KUKA KRL program: PickEsteira.src, PickEsteira.dat

--- PickEsteira.src ---
&ACCESS RVO1
&REL 95
&PARAM DISKPATH = KRC:\R1\Program\MainRoutune\Pick
DEF PickEsteira ( )
   PuxaReceita()
   $Advance=3
   ConfGarra_nowait()

   ;FOLD verifica qual opcao de base para a esteira
      SWITCH PalletAtivo
         CASE 1
            BaseRelativa.X = BaseEsteira1.X + OffsetEsteira1.X
            BaseRelativa.Y = BaseEsteira1.Y + OffsetEsteira1.Y
            BaseRelativa.Z = BaseEsteira1.Z + OffsetEsteira1.Z
            BaseRelativa.A = BaseEsteira1.A + OffsetEsteira1.A
            BaseRelativa.B = BaseEsteira1.B + OffsetEsteira1.B
            BaseRelativa.C = BaseEsteira1.C + OffsetEsteira1.C
         CASE 2
            BaseRelativa.X = BaseEsteira2.X + OffsetEsteira2.X
            BaseRelativa.Y = BaseEsteira2.Y + OffsetEsteira2.Y
            BaseRelativa.Z = BaseEsteira2.Z + OffsetEsteira2.Z
            BaseRelativa.A = BaseEsteira2.A + OffsetEsteira2.A
            BaseRelativa.B = BaseEsteira2.B + OffsetEsteira2.B
            BaseRelativa.C = BaseEsteira2.C + OffsetEsteira2.C
         DEFAULT
            BaseRelativa = NULLFRAME
      ENDSWITCH
   ;ENDFOLD

   ;FOLD PickEsteira de cada receita
      Tpick_esteira()
      XPICK = pick_esteira[PalletAtivo,PickOp]
   ;ENDFOLD

   ;SET BaseRelativa
   $TOOL = TOOL_DATA[1]
   $BASE=BaseRelativa

   ;SET Ponto de pick
   XAPP1PICK = XPICK
   XAPP2PICK = XPICK
   XSAIPICK  = XPICK

   ;Captura o Y da esteira para o ponto de aproximacao
   ;IF (PalletAtivo==1) THEN
   ;   XAPP1PICK.Y = XAPP1PICK.Y - 50
   ;   XAPP2PICK.Y = XAPP2PICK.Y - 50
   ;ENDIF

   ;IF (PalletAtivo==2) THEN
   ;   XAPP1PICK.Y = XAPP1PICK.Y + 50
   ;   XAPP2PICK.Y = XAPP2PICK.Y + 50
   ;ENDIF

   ;FOLD raciocinio do calculo de igualar bases
      ;    ZPick  _      _ ZPlace
      ;           |      |
      ;           |      |
      ;           |      |
      ;           |      - BPlace
      ;           |      |
      ;    BPick  -      |
      ;           |      |
      ;           |      |
      ;             ZERO

      ;ZPick  + BPick  = ZPlace + BPlace

      ;ZPick  = ZPlace + BPlace - BPick
      ;ZPlace = ZPick  + BPick  - BPlace

      ;ALTURATOPO=1800
      ;ZPick  = ALTURATOPO - BPick
      ;ZPlace = ALTURATOPO - BPlace
   ;ENDFOLD

   ;FOLD TOPO DINAMICO IGUALANDO A BASE PLACE COM A DO PICK
      ;Puxa qual o ponto que sera feito o Place
      SetPlacePos()
      ;iguala as bases para obter o Z relativo
      ;ZPick      = ZPlace       +  BPlace                                          - BPick
      XAPP1PICK.Z = XApp1Place.Z + (BasePoint.Z + OffSetPallet.Z + OffsetProduto.Z) - BaseRelativa.Z

      ;Configura a altura de saida do pick
      XSAIPICK.Z = XAPP1PICK.Z

      ;Se o pallet estiver completo o pick eh forcado com a altura MAX
      IF (PalletCompleto==TRUE) THEN
         XAPP1PICK.Z = AlturaPalletCompleto - BaseRelativa.Z
         PalletCompleto=FALSE
      ENDIF

      ;Por seguranca deve garantir que sempre sera acima da altura minima
      ; ZPick2 = ALTURATOPO - BPick
      ; IF (ZPick1 < ZPick2)
      IF (XAPP1PICK.Z<(ALTURATOPO - BaseRelativa.Z)) THEN
         XAPP1PICK.Z = ALTURATOPO - BaseRelativa.Z
      ENDIF
      ;Por seguranca deve garantir que sempre sera acima da altura minima
      IF (XSAIPICK.Z<(ALTURATOPO - BaseRelativa.Z)) THEN
         XSAIPICK.Z  = ALTURATOPO - BaseRelativa.Z
      ENDIF
   ;ENDFOLD

   ;APROXIMA TOPO
   PTP XAPP1PICK C_DIS

   ;CONFIGURA GARRA
   ;ConfGarra()
   ConfGarra_Wait()

   ;APROXIMA DA CAIXA
   LIN XAPP2PICK C_DIS C_DIS

   ;PONTO DE PICK
   LIN XPICK

   ;Fecha Garra
   FechaGarra()

   ;TRAVA/FREIA GARRA
   IF (TravaGarra) THEN
      HomePositionBrake = TRUE
      WorkPositionBrake = FALSE
   ELSE
      HomePositionBrake = FALSE
      WorkPositionBrake = TRUE
   ENDIF

   ;SOBE EM MOVIMENTO RELATIVO
   LIN XSAIPICK

END

--- PickEsteira.dat ---
&ACCESS RVO1
&REL 95
&PARAM DISKPATH = KRC:\R1\Program\MainRoutune\Pick
DEFDAT  PICKESTEIRA
REAL TopoRelativo=707.875305
FRAME RelFrame={X 0.0,Y 0.0,Z 0.0,A 0.0,B 0.0,C 0.0}
FRAME BaseRelativa={X 648.495,Y -1967.36694,Z -56.0000,A 0.0,B 0.0,C 0.0}
DECL E6POS XAPP1PICK={X 491.530762,Y 56.8316116,Z 1968.79492,A 90.0000,B 0.0,C -180.000,S 2,T 34,E1 0.0,E2 0.0,E3 0.0,E4 0.0,E5 0.0,E6 0.0}
DECL E6POS XAPP2PICK={X 491.530762,Y 56.8316116,Z 1343.55737,A 90.0000,B 0.0,C -180.000,S 2,T 34,E1 0.0,E2 0.0,E3 0.0,E4 0.0,E5 0.0,E6 0.0}
DECL E6POS XPICK={X 491.530762,Y 56.8316116,Z 1343.55737,A 90.0000,B 0.0,C -180.000,S 2,T 34,E1 0.0,E2 0.0,E3 0.0,E4 0.0,E5 0.0,E6 0.0}
DECL E6POS XSAIPICK={X 491.530762,Y 56.8316116,Z 1656.00,A 90.0000,B 0.0,C -180.000,S 2,T 34,E1 0.0,E2 0.0,E3 0.0,E4 0.0,E5 0.0,E6 0.0}
;pontos exportados de FURUKAWA
ENDDAT
